   IF "PLC_Signals_DB".CH_NUMBER[0] THEN
       "PLC_Signals_DB".CH_NUMBER[1] := 0;
       "PLC_Signals_DB".CH_NUMBER[2] := 0;
       "PLC_Signals_DB".CH_NUMBER[3] := 0;
       "PLC_Signals_DB".CH_NUMBER[4] := 0;
       "PLC_Signals_DB".CH_NUMBER[5] := 0;
       "PLC_Signals_DB".CH_NUMBER[6] := 0;
       "PLC_Signals_DB".CH_NUMBER[7] := 0;
       "PLC_Signals_DB".CH_NUMBER[8] := 0;
       "PLC_Signals_DB".CH_NUMBER[9] := 0;
       "PLC_Signals_DB".CH_NUMBER[10] := 0;
       "PLC_Signals_DB".CH_NUMBER[11] := 0;
       "PLC_Signals_DB".CH_NUMBER[12] := 0;
       "PLC_Signals_DB".CH_NUMBER[13] := 0;
       "PLC_Signals_DB".CH_NUMBER[14] := 0;
       "PLC_Signals_DB".CH_NUMBER[15] := 0;
       "PLC_Signals_DB".CH_NUMBER[16] := 0;
       "PLC_Signals_DB".CH_NUMBER[17] := 0;
       "PLC_Signals_DB".CH_NUMBER[18] := 0;
       "PLC_Signals_DB".CH_NUMBER[19] := 0;
       "PLC_Signals_DB".CH_NUMBER[20] := 0;

       "DB_TST".CH_NUMBER := 0;
       "DB_TST".CH_NUMBER_OLD := "DB_TST".CH_NUMBER;
       "PLC_Signals_DB".CH_NUMBER[0] := 0;
   END_IF;

   CASE "DB_TST".CH_NUMBER OF
       1:
           IF "DB_TST".CH_NUMBER <> "DB_TST".CH_NUMBER_OLD THEN
               #Config_AI := #AI_2_0;
               "DB_TST".CH_NUMBER_OLD := "DB_TST".CH_NUMBER;
               ;
           END_IF;
           #Config_AI.ING_Value := #AI_2_0.ING_Value;
           #Config_AI.SCALED := #AI_2_0.SCALED;
           #Config_AI.State := #AI_2_0.State;
           #AI_2_0 := #Config_AI;
           ;
       2:
           IF "DB_TST".CH_NUMBER <> "DB_TST".CH_NUMBER_OLD THEN
               #Config_AI := #AI_2_1;
               "DB_TST".CH_NUMBER_OLD := "DB_TST".CH_NUMBER;
               ;
           END_IF;
           #Config_AI.ING_Value := #AI_2_1.ING_Value;
           #Config_AI.SCALED := #AI_2_1.SCALED;
           #Config_AI.State := #AI_2_1.State;
           #AI_2_1 := #Config_AI;
           ;
       3:
          IF "DB_TST".CH_NUMBER <> "DB_TST".CH_NUMBER_OLD THEN
               #Config_AI := #AI_2_2;
               "DB_TST".CH_NUMBER_OLD := "DB_TST".CH_NUMBER;
               ;
           END_IF;
           #Config_AI.ING_Value := #AI_2_2.ING_Value;
           #Config_AI.SCALED := #AI_2_2.SCALED;
           #Config_AI.State := #AI_2_2.State;
           #AI_2_2 := #Config_AI;
           ;
       4:
           IF "DB_TST".CH_NUMBER <> "DB_TST".CH_NUMBER_OLD THEN
               #Config_AI := #AI_2_3;
               "DB_TST".CH_NUMBER_OLD := "DB_TST".CH_NUMBER;
               ;
           END_IF;
           #Config_AI.ING_Value := #AI_2_3.ING_Value;
           #Config_AI.SCALED := #AI_2_3.SCALED;
           #Config_AI.State := #AI_2_3.State;
           #AI_2_3 := #Config_AI;
           ;
       5:
            IF "DB_TST".CH_NUMBER <> "DB_TST".CH_NUMBER_OLD THEN
               #Config_AI := #AI_2_4;
               "DB_TST".CH_NUMBER_OLD := "DB_TST".CH_NUMBER;
               ;
           END_IF;
           #Config_AI.ING_Value := #AI_2_4.ING_Value;
           #Config_AI.SCALED := #AI_2_4.SCALED;
           #Config_AI.State := #AI_2_4.State;
           #AI_2_4 := #Config_AI;
           ;
       6:
          IF "DB_TST".CH_NUMBER <> "DB_TST".CH_NUMBER_OLD THEN
               #Config_AI := #AI_2_5;
               "DB_TST".CH_NUMBER_OLD := "DB_TST".CH_NUMBER;
               ;
           END_IF;
           #Config_AI.ING_Value := #AI_2_5.ING_Value;
           #Config_AI.SCALED := #AI_2_5.SCALED;
           #Config_AI.State := #AI_2_5.State;
           #AI_2_5 := #Config_AI;
           ;
       7:
           IF "DB_TST".CH_NUMBER <> "DB_TST".CH_NUMBER_OLD THEN
               #Config_AI := #AI_2_6;
               "DB_TST".CH_NUMBER_OLD := "DB_TST".CH_NUMBER;
               ;
           END_IF;
           #Config_AI.ING_Value := #AI_2_6.ING_Value;
           #Config_AI.SCALED := #AI_2_6.SCALED;
           #Config_AI.State := #AI_2_6.State;
           #AI_2_6 := #Config_AI;
           ;
       8:
            IF "DB_TST".CH_NUMBER <> "DB_TST".CH_NUMBER_OLD THEN
               #Config_AI := #AI_2_7;
               "DB_TST".CH_NUMBER_OLD := "DB_TST".CH_NUMBER;
               ;
           END_IF;
           #Config_AI.ING_Value := #AI_2_7.ING_Value;
           #Config_AI.SCALED := #AI_2_7.SCALED;
           #Config_AI.State := #AI_2_7.State;
           #AI_2_7 := #Config_AI;
           ;
       9:
           IF "DB_TST".CH_NUMBER <> "DB_TST".CH_NUMBER_OLD THEN
               #Config_AI := #AI_3_0;
               "DB_TST".CH_NUMBER_OLD := "DB_TST".CH_NUMBER;
               ;
           END_IF;
           #Config_AI.ING_Value := #AI_3_0.ING_Value;
           #Config_AI.SCALED := #AI_3_0.SCALED;
           #Config_AI.State := #AI_3_0.State;
           #AI_3_0 := #Config_AI;
           ;
       10:
           IF "DB_TST".CH_NUMBER <> "DB_TST".CH_NUMBER_OLD THEN
               #Config_AI := #AI_3_1;
               "DB_TST".CH_NUMBER_OLD := "DB_TST".CH_NUMBER;
               ;
           END_IF;
           #Config_AI.ING_Value := #AI_3_1.ING_Value;
           #Config_AI.SCALED := #AI_3_1.SCALED;
           #Config_AI.State := #AI_3_1.State;
           #AI_3_1 := #Config_AI;
           ;
       11:
           IF "DB_TST".CH_NUMBER <> "DB_TST".CH_NUMBER_OLD THEN
               #Config_AI := #AI_3_2;
               "DB_TST".CH_NUMBER_OLD := "DB_TST".CH_NUMBER;
               ;
           END_IF;
           #Config_AI.ING_Value := #AI_3_2.ING_Value;
           #Config_AI.SCALED := #AI_3_2.SCALED;
           #Config_AI.State := #AI_3_2.State;
           #AI_3_2 := #Config_AI;
           ;
       12:
           IF "DB_TST".CH_NUMBER <> "DB_TST".CH_NUMBER_OLD THEN
               #Config_AI := #AI_3_3;
               "DB_TST".CH_NUMBER_OLD := "DB_TST".CH_NUMBER;
               ;
           END_IF;
           #Config_AI.ING_Value := #AI_3_3.ING_Value;
           #Config_AI.SCALED := #AI_3_3.SCALED;
           #Config_AI.State := #AI_3_3.State;
           #AI_3_3 := #Config_AI;
           ;
       13:
           IF "DB_TST".CH_NUMBER <> "DB_TST".CH_NUMBER_OLD THEN
               #Config_AI := #AI_3_4;
               "DB_TST".CH_NUMBER_OLD := "DB_TST".CH_NUMBER;
               ;
           END_IF;
           #Config_AI.ING_Value := #AI_3_4.ING_Value;
           #Config_AI.SCALED := #AI_3_4.SCALED;
           #Config_AI.State := #AI_3_4.State;
           #AI_3_4 := #Config_AI;
           ;
       14:
           IF "DB_TST".CH_NUMBER <> "DB_TST".CH_NUMBER_OLD THEN
               #Config_AI := #AI_3_5;
               "DB_TST".CH_NUMBER_OLD := "DB_TST".CH_NUMBER;
               ;
           END_IF;
           #Config_AI.ING_Value := #AI_3_5.ING_Value;
           #Config_AI.SCALED := #AI_3_5.SCALED;
           #Config_AI.State := #AI_3_5.State;
           #AI_3_5 := #Config_AI;
           ;
       15:
           IF "DB_TST".CH_NUMBER <> "DB_TST".CH_NUMBER_OLD THEN
               #Config_AI := #AI_3_6;
               "DB_TST".CH_NUMBER_OLD := "DB_TST".CH_NUMBER;
               ;
           END_IF;
           #Config_AI.ING_Value := #AI_3_6.ING_Value;
           #Config_AI.SCALED := #AI_3_6.SCALED;
           #Config_AI.State := #AI_3_6.State;
           #AI_3_6 := #Config_AI;
           ;
       16:
           IF "DB_TST".CH_NUMBER <> "DB_TST".CH_NUMBER_OLD THEN
               #Config_AI := #AI_3_7;
               "DB_TST".CH_NUMBER_OLD := "DB_TST".CH_NUMBER;
               ;
           END_IF;
           #Config_AI.ING_Value := #AI_3_7.ING_Value;
           #Config_AI.SCALED := #AI_3_7.SCALED;
           #Config_AI.State := #AI_3_7.State;
           #AI_3_7 := #Config_AI;
           ;
       ELSE  // Statement section ELSE
           ;
   END_CASE;
END_FUNCTION

FUNCTION "AI" : Void   // FC24, LAD
{ S7_Optimized_Access := 'TRUE' }
VERSION : 0.1
   VAR_IN_OUT
      AI : Struct   // ????????? ? AI
         Hihi_Value : Real;   // True
         High_Value : Real;   // True
         Low_Value : Real;   // True
         Lolo_Value : Real;   // True
         MIN_Current : Real;   // True
         MAX_Current : Real;   // True
         MAX_Value : Real;   // True
         MIN_Value : Real;   // True
         Underflow_RAW : Real;   // True
         Overflow_RAW : Real;   // True
         SCALED : Real;   // True
         ING_Value : Real;   // True
         Manual_Value : Real;   // True
         Alarm_Delay : Int;   // True
         Warning_Delay : Int;   // True
         AVG_Delay : Real;   // True
         Underflow_Delay : Int;   // True
         Overflow_Delay : Int;   // True
         StateHMI : Int;
         State : Word;   // True
         Modeee : Word;   // True
         bools : Word;   // True
         AI_RAW_MIN : Int;   // True
         AI_RAW_MAX : Int;   // True
         Hihi_EN : Bool;   // True
         High_EN : Bool;   // True
         Low_En : Bool;   // True
         Lolo_EN : Bool;   // True
      END_STRUCT;
      AI_RAW : Int;   // ???????? ??? ?? ?????
      Hihi_TImer : IEC_TIMER;
      High_Timer : IEC_TIMER;
      Low_Timer : IEC_TIMER;
      Lolo_Timer : IEC_TIMER;
      WB_Timer : IEC_TIMER;
      OVerflow_Timer : IEC_TIMER;
   END_VAR
   VAR_TEMP
      Hihi_Int : Bool;   // ????????????? ???????????? ??????? Hihi ??? ?????????? ???????? ?????????
      High_Int : Bool;   // ????????????? ???????????? ??????? High ??? ?????????? ???????? ?????????
      Low_Int : Bool;   // ????????????? ???????????? ??????? Low ??? ?????????? ???????? ?????????
      Lolo_Int : Bool;   // ????????????? ???????????? ??????? Lolo ??? ?????????? ???????? ?????????
      Scaled_4_20mA : Real;   // ???????? ???? ?? ?????, ???????????????? ? 4-20??
      WB_Int : Bool;   // ????????????? ????????????? ?????? ???????
      Last_value : Real;   // ???????? ??? FailSafe_Mode
      count : Int;   // ?????????? ???????? ??? ??????????
      time_int : Int;   // ????? ? INT
      current_count : Int;   // ??????? ?????????? ???????? ??? ??????????
      summ_AVG_Value : Real;   // ????? ???????? ??? ??????????
      tmp_scaled : Real;   // ???????????????? ???????? ??? ??????????
      Overflow_int : Bool;   // ??????????????? ???????????? ????????????? ??????? <
      Underflow_int : Bool;   // ??????????????? ???????????? ????????????? ??????? >
      AVG_Delay_real : Real;
      Alarm_Delay_int : Time;
      Warning_Delay_int : Time;
      Underflow_Delay_int : Time;
      Overflow_Delay_int : Time;
      TMP_ING_Value : Real;
      et1 : Time;
      et2 : Time;
      et3 : Time;
      et4 : Time;
      et5 : Time;
      et6 : Time;
      ust_avg_up : Real;
      ust_avg_down : Real;
   END_VAR
   VAR CONSTANT
      AI_Time : Int := 250;   // ????? ?????? AI (??)
   END_VAR
   VAR_TEMP   // added for the SCL form of the ladder/FBD networks
      _w1 : Bool;
      _w2 : Bool;
      _w3 : Bool;
      _w4 : Bool;
      _w5 : Bool;
      _w6 : Bool;
      _w7 : Bool;
      _w8 : Bool;
      _w9 : Bool;
      _w10 : Bool;
      _w11 : Bool;
      _w12 : Bool;
      _w13 : Bool;
      _w14 : Bool;
      _w15 : Bool;
   END_VAR
BEGIN

REGION Network 1: Пересчет времени
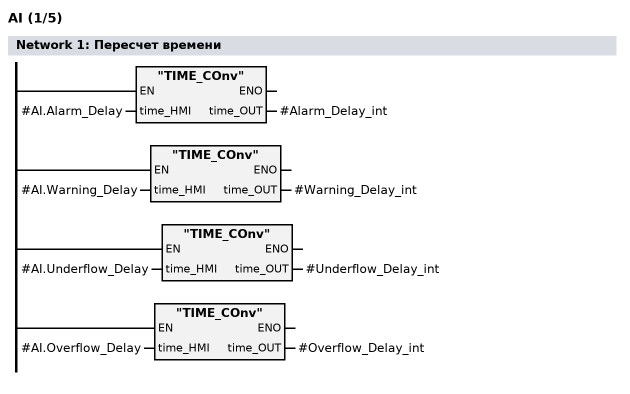
   RUNG wire#powerrail
      "TIME_COnv"(time_HMI := #AI.Alarm_Delay, time_OUT => #Alarm_Delay_int)
   END_RUNG
   RUNG wire#powerrail
      "TIME_COnv"(time_HMI := #AI.Warning_Delay, time_OUT => #Warning_Delay_int)
   END_RUNG
   RUNG wire#powerrail
      "TIME_COnv"(time_HMI := #AI.Underflow_Delay, time_OUT => #Underflow_Delay_int)
   END_RUNG
   RUNG wire#powerrail
      "TIME_COnv"(time_HMI := #AI.Overflow_Delay, time_OUT => #Overflow_Delay_int)
   END_RUNG
   // the same network as SCL:
   "TIME_COnv"(time_HMI := #AI.Alarm_Delay, time_OUT => #Alarm_Delay_int);
   "TIME_COnv"(time_HMI := #AI.Warning_Delay, time_OUT => #Warning_Delay_int);
   "TIME_COnv"(time_HMI := #AI.Underflow_Delay, time_OUT => #Underflow_Delay_int);
   "TIME_COnv"(time_HMI := #AI.Overflow_Delay, time_OUT => #Overflow_Delay_int);
END_REGION

REGION Network 2: авто конвертация в инж. и физ. значение
   // Автоматическая обработка сигналов
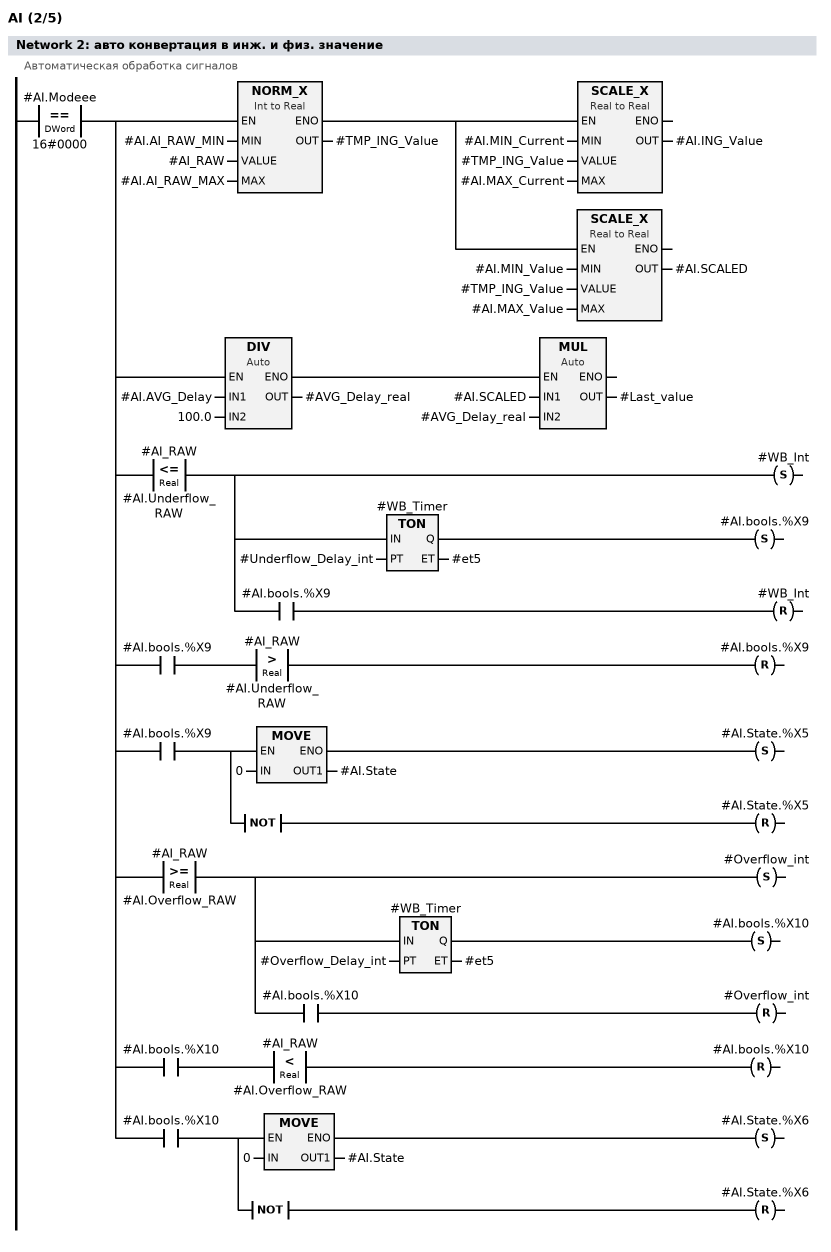
   // ENO of a box is taken as its EN; it also drops when the box reports an error
   #_w1 := #AI.Modeee = 16#0000;
   IF #_w1 THEN
       #TMP_ING_Value := NORM_X(MIN := #AI.AI_RAW_MIN, VALUE := #AI_RAW, MAX := #AI.AI_RAW_MAX);
       #AI.ING_Value := SCALE_X(MIN := #AI.MIN_Current, VALUE := #TMP_ING_Value, MAX := #AI.MAX_Current);
       #AI.SCALED := SCALE_X(MIN := #AI.MIN_Value, VALUE := #TMP_ING_Value, MAX := #AI.MAX_Value);
       #AVG_Delay_real := #AI.AVG_Delay / 100.0;
       #Last_value := #AI.SCALED * #AVG_Delay_real;
   END_IF;
   #_w2 := #_w1 AND (#AI_RAW <= #AI.Underflow_RAW);
   IF #_w2 THEN #WB_Int := TRUE; END_IF;
   #WB_Timer.TON(IN := #_w2, PT := #Underflow_Delay_int, ET => #et5);
   IF #WB_Timer.Q THEN #AI.bools.%X9 := TRUE; END_IF;
   IF #_w2 AND #AI.bools.%X9 THEN #WB_Int := FALSE; END_IF;
   IF #_w1 AND #AI.bools.%X9 AND (#AI_RAW > #AI.Underflow_RAW) THEN #AI.bools.%X9 := FALSE; END_IF;
   #_w3 := #_w1 AND #AI.bools.%X9;
   IF #_w3 THEN
       #AI.State := 0;
       #AI.State.%X5 := TRUE;
   END_IF;
   IF NOT #_w3 THEN #AI.State.%X5 := FALSE; END_IF;
   #_w4 := #_w1 AND (#AI_RAW >= #AI.Overflow_RAW);
   IF #_w4 THEN #Overflow_int := TRUE; END_IF;
   #WB_Timer.TON(IN := #_w4, PT := #Overflow_Delay_int, ET => #et5);
   IF #WB_Timer.Q THEN #AI.bools.%X10 := TRUE; END_IF;
   IF #_w4 AND #AI.bools.%X10 THEN #Overflow_int := FALSE; END_IF;
   IF #_w1 AND #AI.bools.%X10 AND (#AI_RAW < #AI.Overflow_RAW) THEN #AI.bools.%X10 := FALSE; END_IF;
   #_w5 := #_w1 AND #AI.bools.%X10;
   IF #_w5 THEN
       #AI.State := 0;
       #AI.State.%X6 := TRUE;
   END_IF;
   IF NOT #_w5 THEN #AI.State.%X6 := FALSE; END_IF;
END_REGION

REGION Network 3: ручной ввод и ремонт, при это ток вседа равен 4мА, чтобы обрыв не вылетал
   // ремонт или ручной ввод
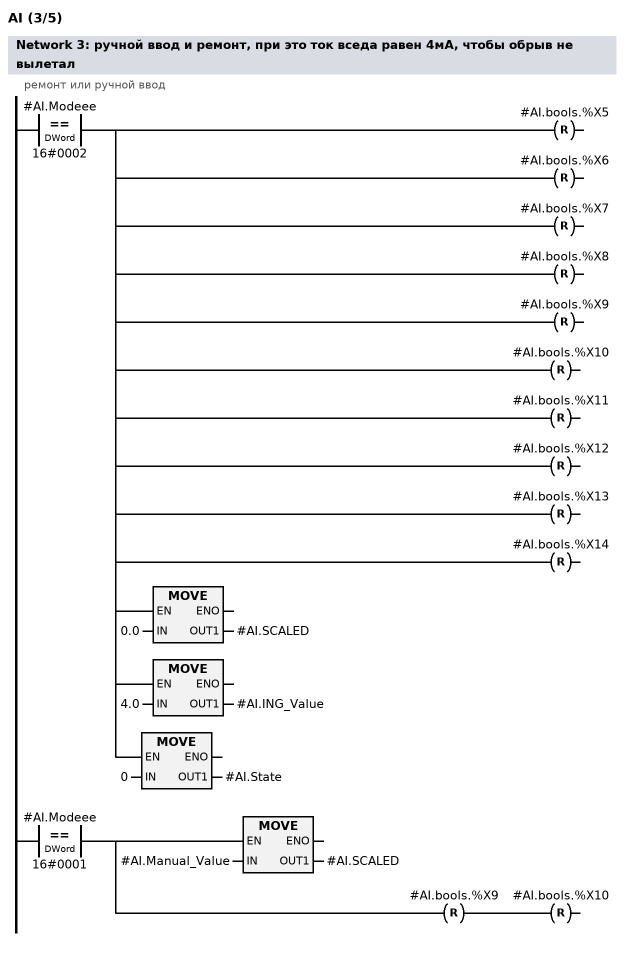
   RUNG wire#powerrail
      { S7_Templates := "SrcType := DWord" } EQ_Contact(in1 := #AI.Modeee, in2 := 16#0002)
      wire#w1
      R_Coil( #AI.bools.%X5 )
   END_RUNG
   RUNG wire#w1
      R_Coil( #AI.bools.%X6 )
   END_RUNG
   RUNG wire#w1
      R_Coil( #AI.bools.%X7 )
   END_RUNG
   RUNG wire#w1
      R_Coil( #AI.bools.%X8 )
   END_RUNG
   RUNG wire#w1
      R_Coil( #AI.bools.%X9 )
   END_RUNG
   RUNG wire#w1
      R_Coil( #AI.bools.%X10 )
   END_RUNG
   RUNG wire#w1
      R_Coil( #AI.bools.%X11 )
   END_RUNG
   RUNG wire#w1
      R_Coil( #AI.bools.%X12 )
   END_RUNG
   RUNG wire#w1
      R_Coil( #AI.bools.%X13 )
   END_RUNG
   RUNG wire#w1
      R_Coil( #AI.bools.%X14 )
   END_RUNG
   RUNG wire#w1
      { S7_GenerateENO := "TRUE" } Move(in := 0.0, out1 => #AI.SCALED)
   END_RUNG
   RUNG wire#w1
      { S7_GenerateENO := "TRUE" } Move(in := 4.0, out1 => #AI.ING_Value)
   END_RUNG
   RUNG wire#w1
      { S7_GenerateENO := "TRUE" } Move(in := 0, out1 => #AI.State)
   END_RUNG
   RUNG wire#powerrail
      { S7_Templates := "SrcType := DWord" } EQ_Contact(in1 := #AI.Modeee, in2 := 16#0001)
      wire#w2
      { S7_GenerateENO := "TRUE" } Move(in := #AI.Manual_Value, out1 => #AI.SCALED)
   END_RUNG
   RUNG wire#w2
      R_Coil( #AI.bools.%X9 )
      R_Coil( #AI.bools.%X10 )
   END_RUNG
   // the same network as SCL:
   IF #AI.Modeee = 16#0002 THEN
       #AI.bools.%X5 := FALSE;
       #AI.bools.%X6 := FALSE;
       #AI.bools.%X7 := FALSE;
       #AI.bools.%X8 := FALSE;
       #AI.bools.%X9 := FALSE;
       #AI.bools.%X10 := FALSE;
       #AI.bools.%X11 := FALSE;
       #AI.bools.%X12 := FALSE;
       #AI.bools.%X13 := FALSE;
       #AI.bools.%X14 := FALSE;
       #AI.SCALED := 0.0;
       #AI.ING_Value := 4.0;
       #AI.State := 0;
   END_IF;
   IF #AI.Modeee = 16#0001 THEN
       #AI.SCALED := #AI.Manual_Value;
       #AI.bools.%X9 := FALSE;
       #AI.bools.%X10 := FALSE;
   END_IF;
END_REGION

REGION Network 4: уставки
   // Автоматическая обработка сигналов
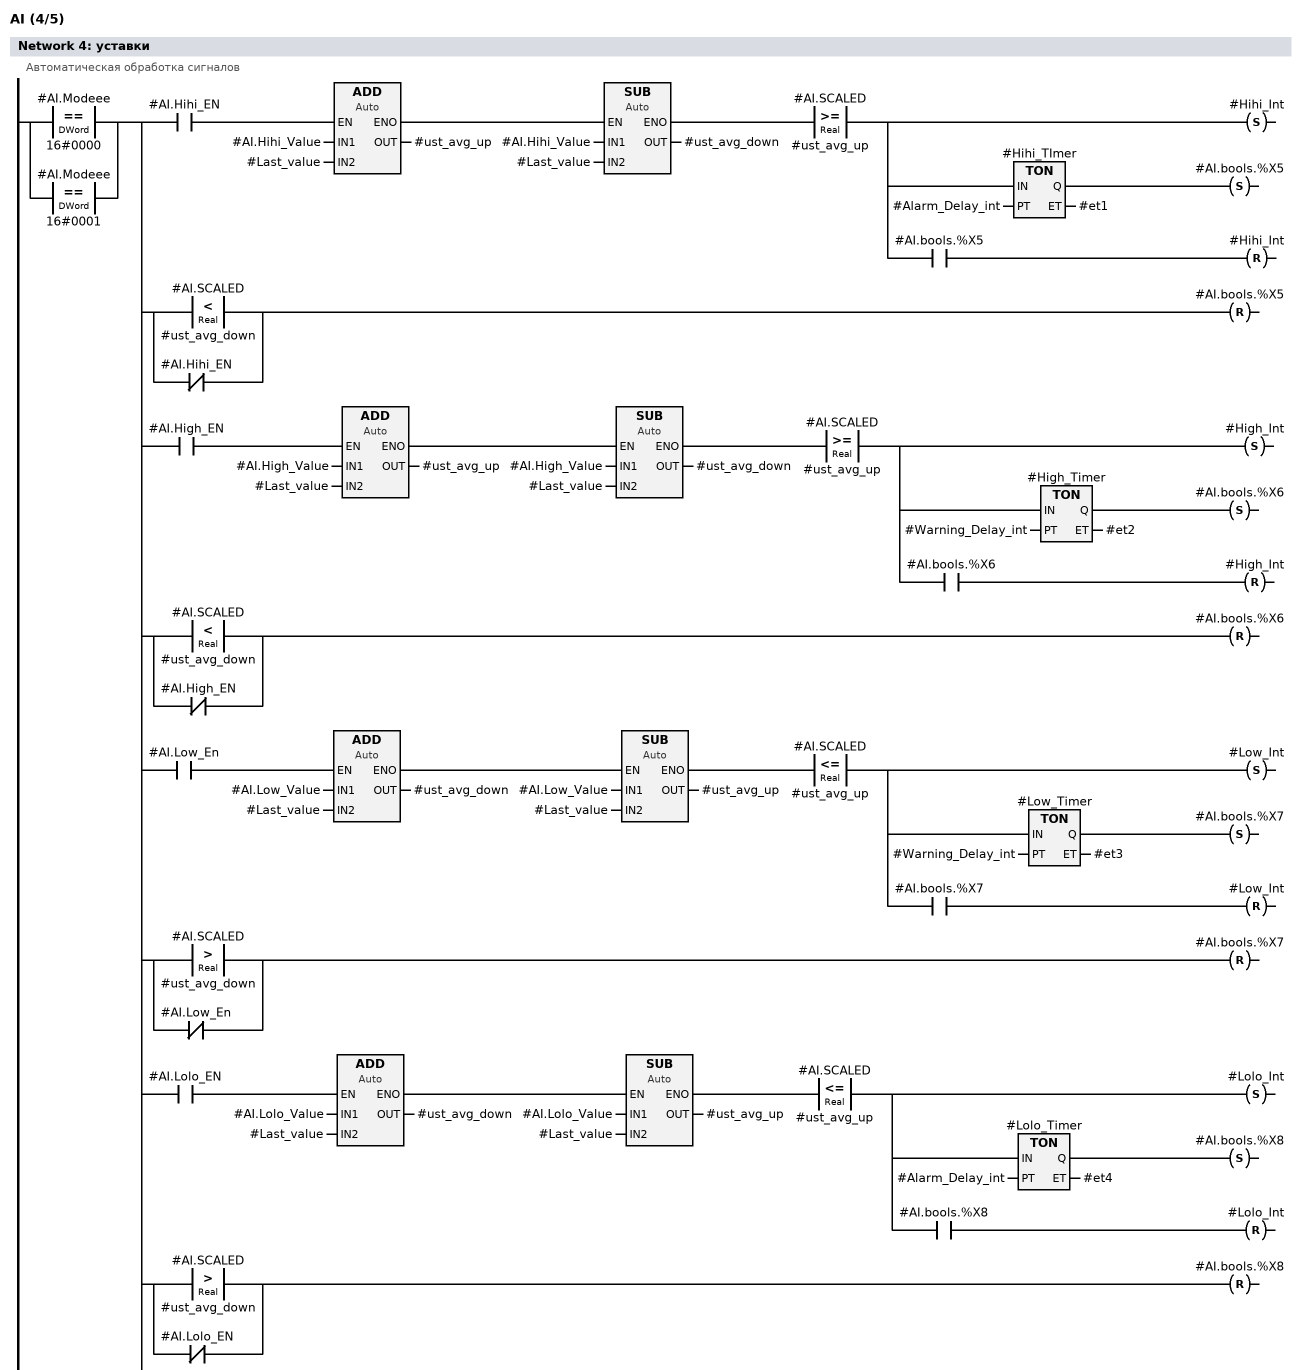
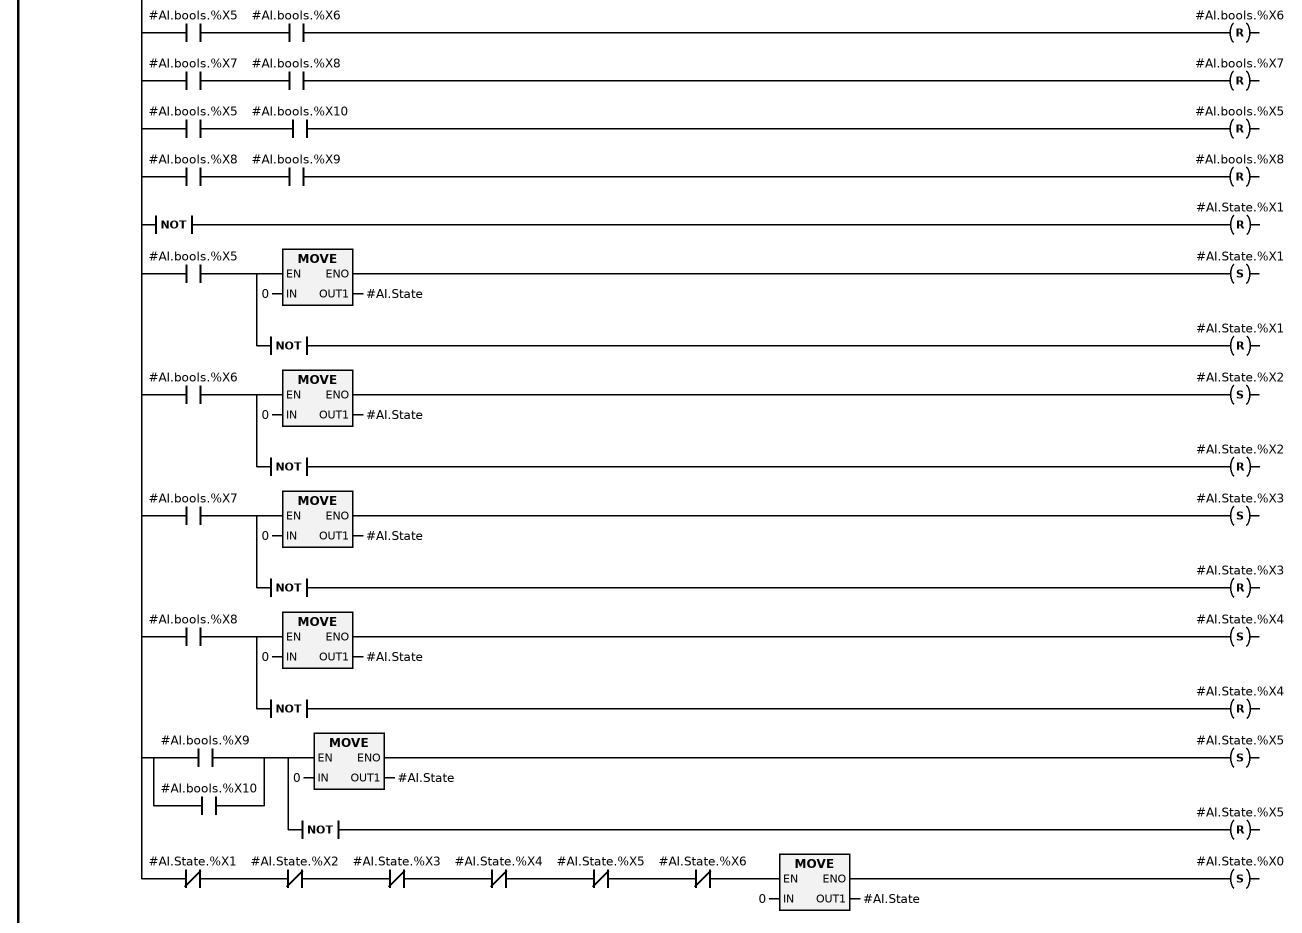
   // ENO of a box is taken as its EN; it also drops when the box reports an error
   #_w1 := (#AI.Modeee = 16#0000) OR (#AI.Modeee = 16#0001);
   #_w2 := #_w1 AND #AI.Hihi_EN;
   IF #_w2 THEN
       #ust_avg_up := #AI.Hihi_Value + #Last_value;
       #ust_avg_down := #AI.Hihi_Value - #Last_value;
   END_IF;
   #_w3 := #_w2 AND (#AI.SCALED >= #ust_avg_up);
   IF #_w3 THEN #Hihi_Int := TRUE; END_IF;
   #Hihi_TImer.TON(IN := #_w3, PT := #Alarm_Delay_int, ET => #et1);
   IF #Hihi_TImer.Q THEN #AI.bools.%X5 := TRUE; END_IF;
   IF #_w3 AND #AI.bools.%X5 THEN #Hihi_Int := FALSE; END_IF;
   IF #_w1 AND ((#AI.SCALED < #ust_avg_down) OR NOT #AI.Hihi_EN) THEN #AI.bools.%X5 := FALSE; END_IF;
   #_w4 := #_w1 AND #AI.High_EN;
   IF #_w4 THEN
       #ust_avg_up := #AI.High_Value + #Last_value;
       #ust_avg_down := #AI.High_Value - #Last_value;
   END_IF;
   #_w5 := #_w4 AND (#AI.SCALED >= #ust_avg_up);
   IF #_w5 THEN #High_Int := TRUE; END_IF;
   #High_Timer.TON(IN := #_w5, PT := #Warning_Delay_int, ET => #et2);
   IF #High_Timer.Q THEN #AI.bools.%X6 := TRUE; END_IF;
   IF #_w5 AND #AI.bools.%X6 THEN #High_Int := FALSE; END_IF;
   IF #_w1 AND ((#AI.SCALED < #ust_avg_down) OR NOT #AI.High_EN) THEN #AI.bools.%X6 := FALSE; END_IF;
   #_w6 := #_w1 AND #AI.Low_En;
   IF #_w6 THEN
       #ust_avg_down := #AI.Low_Value + #Last_value;
       #ust_avg_up := #AI.Low_Value - #Last_value;
   END_IF;
   #_w7 := #_w6 AND (#AI.SCALED <= #ust_avg_up);
   IF #_w7 THEN #Low_Int := TRUE; END_IF;
   #Low_Timer.TON(IN := #_w7, PT := #Warning_Delay_int, ET => #et3);
   IF #Low_Timer.Q THEN #AI.bools.%X7 := TRUE; END_IF;
   IF #_w7 AND #AI.bools.%X7 THEN #Low_Int := FALSE; END_IF;
   IF #_w1 AND ((#AI.SCALED > #ust_avg_down) OR NOT #AI.Low_En) THEN #AI.bools.%X7 := FALSE; END_IF;
   #_w8 := #_w1 AND #AI.Lolo_EN;
   IF #_w8 THEN
       #ust_avg_down := #AI.Lolo_Value + #Last_value;
       #ust_avg_up := #AI.Lolo_Value - #Last_value;
   END_IF;
   #_w9 := #_w8 AND (#AI.SCALED <= #ust_avg_up);
   IF #_w9 THEN #Lolo_Int := TRUE; END_IF;
   #Lolo_Timer.TON(IN := #_w9, PT := #Alarm_Delay_int, ET => #et4);
   IF #Lolo_Timer.Q THEN #AI.bools.%X8 := TRUE; END_IF;
   IF #_w9 AND #AI.bools.%X8 THEN #Lolo_Int := FALSE; END_IF;
   IF #_w1 AND ((#AI.SCALED > #ust_avg_down) OR NOT #AI.Lolo_EN) THEN #AI.bools.%X8 := FALSE; END_IF;
   IF #_w1 AND #AI.bools.%X5 AND #AI.bools.%X6 THEN #AI.bools.%X6 := FALSE; END_IF;
   IF #_w1 AND #AI.bools.%X7 AND #AI.bools.%X8 THEN #AI.bools.%X7 := FALSE; END_IF;
   IF #_w1 AND #AI.bools.%X5 AND #AI.bools.%X10 THEN #AI.bools.%X5 := FALSE; END_IF;
   IF #_w1 AND #AI.bools.%X8 AND #AI.bools.%X9 THEN #AI.bools.%X8 := FALSE; END_IF;
   IF NOT #_w1 THEN #AI.State.%X1 := FALSE; END_IF;
   #_w10 := #_w1 AND #AI.bools.%X5;
   IF #_w10 THEN
       #AI.State := 0;
       #AI.State.%X1 := TRUE;
   END_IF;
   IF NOT #_w10 THEN #AI.State.%X1 := FALSE; END_IF;
   #_w11 := #_w1 AND #AI.bools.%X6;
   IF #_w11 THEN
       #AI.State := 0;
       #AI.State.%X2 := TRUE;
   END_IF;
   IF NOT #_w11 THEN #AI.State.%X2 := FALSE; END_IF;
   #_w12 := #_w1 AND #AI.bools.%X7;
   IF #_w12 THEN
       #AI.State := 0;
       #AI.State.%X3 := TRUE;
   END_IF;
   IF NOT #_w12 THEN #AI.State.%X3 := FALSE; END_IF;
   #_w13 := #_w1 AND #AI.bools.%X8;
   IF #_w13 THEN
       #AI.State := 0;
       #AI.State.%X4 := TRUE;
   END_IF;
   IF NOT #_w13 THEN #AI.State.%X4 := FALSE; END_IF;
   #_w14 := #_w1 AND (#AI.bools.%X9 OR #AI.bools.%X10);
   IF #_w14 THEN
       #AI.State := 0;
       #AI.State.%X5 := TRUE;
   END_IF;
   IF NOT #_w14 THEN #AI.State.%X5 := FALSE; END_IF;
   #_w15 := #_w1 AND NOT #AI.State.%X1 AND NOT #AI.State.%X2 AND NOT #AI.State.%X3 AND NOT #AI.State.%X4 AND NOT #AI.State.%X5 AND NOT #AI.State.%X6;
   IF #_w15 THEN
       #AI.State := 0;
       #AI.State.%X0 := TRUE;
   END_IF;
END_REGION

REGION Network 5
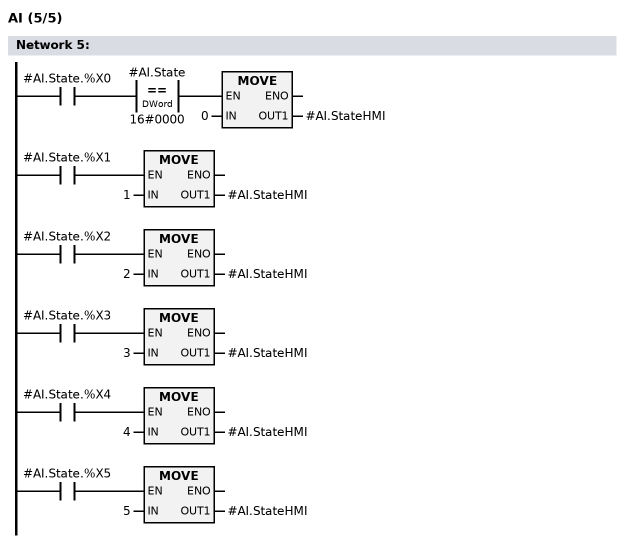
   RUNG wire#powerrail
      Contact( #AI.State.%X0 )
      { S7_Templates := "SrcType := DWord" } EQ_Contact(in1 := #AI.State, in2 := 16#0000)
      Move(in := 0, out1 => #AI.StateHMI)
   END_RUNG
   RUNG wire#powerrail
      Contact( #AI.State.%X1 )
      Move(in := 1, out1 => #AI.StateHMI)
   END_RUNG
   RUNG wire#powerrail
      Contact( #AI.State.%X2 )
      Move(in := 2, out1 => #AI.StateHMI)
   END_RUNG
   RUNG wire#powerrail
      Contact( #AI.State.%X3 )
      Move(in := 3, out1 => #AI.StateHMI)
   END_RUNG
   RUNG wire#powerrail
      Contact( #AI.State.%X4 )
      Move(in := 4, out1 => #AI.StateHMI)
   END_RUNG
   RUNG wire#powerrail
      Contact( #AI.State.%X5 )
      Move(in := 5, out1 => #AI.StateHMI)
   END_RUNG
   // the same network as SCL:
   IF #AI.State.%X0 AND (#AI.State = 16#0000) THEN #AI.StateHMI := 0; END_IF;
   IF #AI.State.%X1 THEN #AI.StateHMI := 1; END_IF;
   IF #AI.State.%X2 THEN #AI.StateHMI := 2; END_IF;
   IF #AI.State.%X3 THEN #AI.StateHMI := 3; END_IF;
   IF #AI.State.%X4 THEN #AI.StateHMI := 4; END_IF;
   IF #AI.State.%X5 THEN #AI.StateHMI := 5; END_IF;
END_REGION
END_FUNCTION

FUNCTION "TIME_COnv" : Void   // FC26, SCL
{ S7_Optimized_Access := 'TRUE' }
VERSION : 0.1
   VAR_INPUT
      time_HMI : Int;
   END_VAR
   VAR_OUTPUT
      time_OUT : Time;
   END_VAR
   VAR_TEMP
      "DINT" : DInt;
      t_DINT : DInt;
   END_VAR
BEGIN
   #t_DINT := INT_TO_DINT(#time_HMI);
   #"DINT" := #t_DINT * 1000;

   #time_OUT := T_CONV(#"DINT");
END_FUNCTION

ORGANIZATION_BLOCK "Main"   // OB1, LAD, ProgramCycle
TITLE = "Main Program Sweep (Cycle)"
{ S7_Optimized_Access := 'TRUE' }
VERSION : 0.1
   VAR_INPUT
      Initial_Call : Bool;   // Initial call of this OB
      Remanence : Bool;   // =True, if remanent data are available
   END_VAR
   VAR_TEMP
      alarm_nmsh : Bool;
      zp_nmsh : Bool;
      alarm_nd_1 : Bool;
      zp_nd_1 : Bool;
      alarm_nd_2 : Bool;
      zp_nd_2 : Bool;
   END_VAR
   VAR_TEMP   // added for the SCL form of the ladder/FBD networks
      _w1 : Bool;
   END_VAR
BEGIN

REGION Network 1: Настройка аналогов с панели
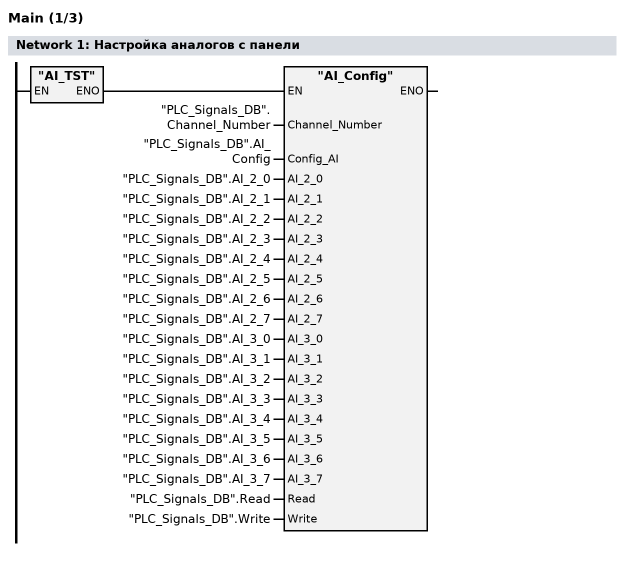
   RUNG wire#powerrail
      "AI_TST"()
      "AI_Config"(Channel_Number := "PLC_Signals_DB".Channel_Number, Config_AI := "PLC_Signals_DB".AI_Config, AI_2_0 := "PLC_Signals_DB".AI_2_0, AI_2_1 := "PLC_Signals_DB".AI_2_1, AI_2_2 := "PLC_Signals_DB".AI_2_2, AI_2_3 := "PLC_Signals_DB".AI_2_3, AI_2_4 := "PLC_Signals_DB".AI_2_4, AI_2_5 := "PLC_Signals_DB".AI_2_5, AI_2_6 := "PLC_Signals_DB".AI_2_6, AI_2_7 := "PLC_Signals_DB".AI_2_7, AI_3_0 := "PLC_Signals_DB".AI_3_0, AI_3_1 := "PLC_Signals_DB".AI_3_1, AI_3_2 := "PLC_Signals_DB".AI_3_2, AI_3_3 := "PLC_Signals_DB".AI_3_3, AI_3_4 := "PLC_Signals_DB".AI_3_4, AI_3_5 := "PLC_Signals_DB".AI_3_5, AI_3_6 := "PLC_Signals_DB".AI_3_6, AI_3_7 := "PLC_Signals_DB".AI_3_7, Read := "PLC_Signals_DB".Read, Write := "PLC_Signals_DB".Write)
   END_RUNG
   // the same network as SCL:
   "AI_TST"(ENO => #_w1);
   IF #_w1 THEN
       "AI_Config"(Channel_Number := "PLC_Signals_DB".Channel_Number,
                   Config_AI := "PLC_Signals_DB".AI_Config,
                   AI_2_0 := "PLC_Signals_DB".AI_2_0,
                   AI_2_1 := "PLC_Signals_DB".AI_2_1,
                   AI_2_2 := "PLC_Signals_DB".AI_2_2,
                   AI_2_3 := "PLC_Signals_DB".AI_2_3,
                   AI_2_4 := "PLC_Signals_DB".AI_2_4,
                   AI_2_5 := "PLC_Signals_DB".AI_2_5,
                   AI_2_6 := "PLC_Signals_DB".AI_2_6,
                   AI_2_7 := "PLC_Signals_DB".AI_2_7,
                   AI_3_0 := "PLC_Signals_DB".AI_3_0,
                   AI_3_1 := "PLC_Signals_DB".AI_3_1,
                   AI_3_2 := "PLC_Signals_DB".AI_3_2,
                   AI_3_3 := "PLC_Signals_DB".AI_3_3,
                   AI_3_4 := "PLC_Signals_DB".AI_3_4,
                   AI_3_5 := "PLC_Signals_DB".AI_3_5,
                   AI_3_6 := "PLC_Signals_DB".AI_3_6,
                   AI_3_7 := "PLC_Signals_DB".AI_3_7,
                   Read := "PLC_Signals_DB".Read,
                   Write := "PLC_Signals_DB".Write);
   END_IF;
END_REGION

REGION Network 2: Горелка
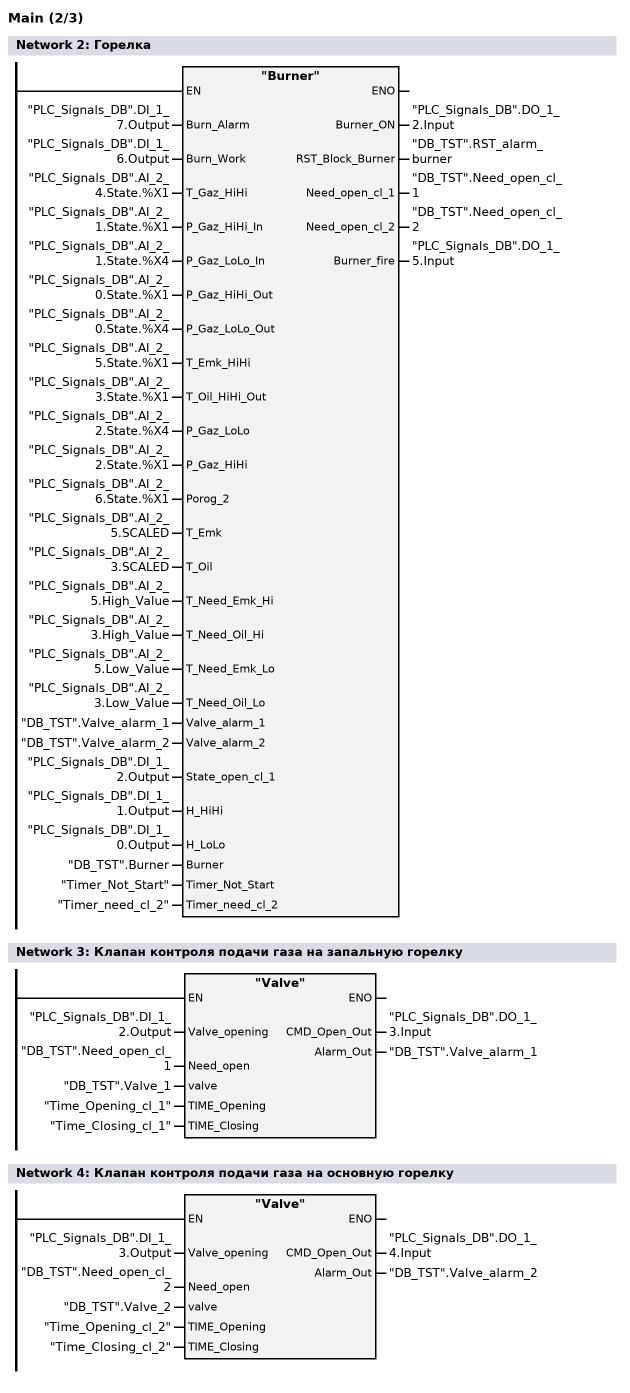
   RUNG wire#powerrail
      "Burner"(Burn_Alarm := "PLC_Signals_DB".DI_1_7.Output, Burn_Work := "PLC_Signals_DB".DI_1_6.Output, T_Gaz_HiHi := "PLC_Signals_DB".AI_2_4.State.%X1, P_Gaz_HiHi_In := "PLC_Signals_DB".AI_2_1.State.%X1, P_Gaz_LoLo_In := "PLC_Signals_DB".AI_2_1.State.%X4, P_Gaz_HiHi_Out := "PLC_Signals_DB".AI_2_0.State.%X1, P_Gaz_LoLo_Out := "PLC_Signals_DB".AI_2_0.State.%X4, T_Emk_HiHi := "PLC_Signals_DB".AI_2_5.State.%X1, T_Oil_HiHi_Out := "PLC_Signals_DB".AI_2_3.State.%X1, P_Gaz_LoLo := "PLC_Signals_DB".AI_2_2.State.%X4, P_Gaz_HiHi := "PLC_Signals_DB".AI_2_2.State.%X1, Porog_2 := "PLC_Signals_DB".AI_2_6.State.%X1, T_Emk := "PLC_Signals_DB".AI_2_5.SCALED, T_Oil := "PLC_Signals_DB".AI_2_3.SCALED, T_Need_Emk_Hi := "PLC_Signals_DB".AI_2_5.High_Value, T_Need_Oil_Hi := "PLC_Signals_DB".AI_2_3.High_Value, T_Need_Emk_Lo := "PLC_Signals_DB".AI_2_5.Low_Value, T_Need_Oil_Lo := "PLC_Signals_DB".AI_2_3.Low_Value, Valve_alarm_1 := "DB_TST".Valve_alarm_1, Valve_alarm_2 := "DB_TST".Valve_alarm_2, State_open_cl_1 := "PLC_Signals_DB".DI_1_2.Output, H_HiHi := "PLC_Signals_DB".DI_1_1.Output, H_LoLo := "PLC_Signals_DB".DI_1_0.Output, Burner := "DB_TST".Burner, Timer_Not_Start := "Timer_Not_Start", Timer_need_cl_2 := "Timer_need_cl_2", Burner_ON => "PLC_Signals_DB".DO_1_2.Input, RST_Block_Burner => "DB_TST".RST_alarm_burner, Need_open_cl_1 => "DB_TST".Need_open_cl_1, Need_open_cl_2 => "DB_TST".Need_open_cl_2, Burner_fire => "PLC_Signals_DB".DO_1_5.Input)
   END_RUNG
   // the same network as SCL:
   "Burner"(Burn_Alarm := "PLC_Signals_DB".DI_1_7.Output,
            Burn_Work := "PLC_Signals_DB".DI_1_6.Output,
            T_Gaz_HiHi := "PLC_Signals_DB".AI_2_4.State.%X1,
            P_Gaz_HiHi_In := "PLC_Signals_DB".AI_2_1.State.%X1,
            P_Gaz_LoLo_In := "PLC_Signals_DB".AI_2_1.State.%X4,
            P_Gaz_HiHi_Out := "PLC_Signals_DB".AI_2_0.State.%X1,
            P_Gaz_LoLo_Out := "PLC_Signals_DB".AI_2_0.State.%X4,
            T_Emk_HiHi := "PLC_Signals_DB".AI_2_5.State.%X1,
            T_Oil_HiHi_Out := "PLC_Signals_DB".AI_2_3.State.%X1,
            P_Gaz_LoLo := "PLC_Signals_DB".AI_2_2.State.%X4,
            P_Gaz_HiHi := "PLC_Signals_DB".AI_2_2.State.%X1,
            Porog_2 := "PLC_Signals_DB".AI_2_6.State.%X1,
            T_Emk := "PLC_Signals_DB".AI_2_5.SCALED,
            T_Oil := "PLC_Signals_DB".AI_2_3.SCALED,
            T_Need_Emk_Hi := "PLC_Signals_DB".AI_2_5.High_Value,
            T_Need_Oil_Hi := "PLC_Signals_DB".AI_2_3.High_Value,
            T_Need_Emk_Lo := "PLC_Signals_DB".AI_2_5.Low_Value,
            T_Need_Oil_Lo := "PLC_Signals_DB".AI_2_3.Low_Value,
            Valve_alarm_1 := "DB_TST".Valve_alarm_1,
            Valve_alarm_2 := "DB_TST".Valve_alarm_2,
            State_open_cl_1 := "PLC_Signals_DB".DI_1_2.Output,
            H_HiHi := "PLC_Signals_DB".DI_1_1.Output,
            H_LoLo := "PLC_Signals_DB".DI_1_0.Output,
            Burner := "DB_TST".Burner,
            Timer_Not_Start := "Timer_Not_Start",
            Timer_need_cl_2 := "Timer_need_cl_2",
            Burner_ON => "PLC_Signals_DB".DO_1_2.Input,
            RST_Block_Burner => "DB_TST".RST_alarm_burner,
            Need_open_cl_1 => "DB_TST".Need_open_cl_1,
            Need_open_cl_2 => "DB_TST".Need_open_cl_2,
            Burner_fire => "PLC_Signals_DB".DO_1_5.Input);
END_REGION

REGION Network 3: Клапан контроля подачи газа на запальную горелку
   RUNG wire#powerrail
      "Valve"(Valve_opening := "PLC_Signals_DB".DI_1_2.Output, Need_open := "DB_TST".Need_open_cl_1, valve := "DB_TST".Valve_1, TIME_Opening := "Time_Opening_cl_1", TIME_Closing := "Time_Closing_cl_1", CMD_Open_Out => "PLC_Signals_DB".DO_1_3.Input, Alarm_Out => "DB_TST".Valve_alarm_1)
   END_RUNG
   // the same network as SCL:
   "Valve"(Valve_opening := "PLC_Signals_DB".DI_1_2.Output,
           Need_open := "DB_TST".Need_open_cl_1,
           valve := "DB_TST".Valve_1,
           TIME_Opening := "Time_Opening_cl_1",
           TIME_Closing := "Time_Closing_cl_1",
           CMD_Open_Out => "PLC_Signals_DB".DO_1_3.Input,
           Alarm_Out => "DB_TST".Valve_alarm_1);
END_REGION

REGION Network 4: Клапан контроля подачи газа на основную горелку
   RUNG wire#powerrail
      "Valve"(Valve_opening := "PLC_Signals_DB".DI_1_3.Output, Need_open := "DB_TST".Need_open_cl_2, valve := "DB_TST".Valve_2, TIME_Opening := "Time_Opening_cl_2", TIME_Closing := "Time_Closing_cl_2", CMD_Open_Out => "PLC_Signals_DB".DO_1_4.Input, Alarm_Out => "DB_TST".Valve_alarm_2)
   END_RUNG
   // the same network as SCL:
   "Valve"(Valve_opening := "PLC_Signals_DB".DI_1_3.Output,
           Need_open := "DB_TST".Need_open_cl_2,
           valve := "DB_TST".Valve_2,
           TIME_Opening := "Time_Opening_cl_2",
           TIME_Closing := "Time_Closing_cl_2",
           CMD_Open_Out => "PLC_Signals_DB".DO_1_4.Input,
           Alarm_Out => "DB_TST".Valve_alarm_2);
END_REGION

REGION Network 5: MB_Comm_Load_DB
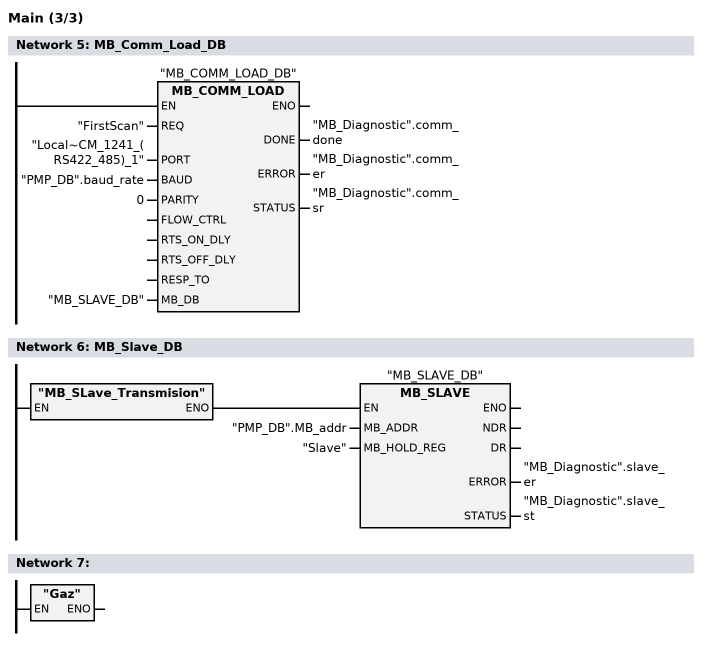
   "MB_COMM_LOAD_DB"(REQ := "FirstScan",   // MB_COMM_LOAD
                     PORT := "Local~CM_1241_(RS422_485)_1",
                     BAUD := "PMP_DB".baud_rate,
                     PARITY := 0,
                     MB_DB := "MB_SLAVE_DB",
                     DONE => "MB_Diagnostic".comm_done,
                     ERROR => "MB_Diagnostic".comm_er,
                     STATUS => "MB_Diagnostic".comm_sr);
END_REGION

REGION Network 6: MB_Slave_DB
   "MB_SLave_Transmision"(ENO => #_w1);
   IF #_w1 THEN
       "MB_SLAVE_DB"(MB_ADDR := "PMP_DB".MB_addr,   // MB_SLAVE
                     MB_HOLD_REG := "Slave",
                     ERROR => "MB_Diagnostic".slave_er,
                     STATUS => "MB_Diagnostic".slave_st);
   END_IF;
END_REGION

REGION Network 7
   RUNG wire#powerrail
      "Gaz"()
   END_RUNG
   // the same network as SCL:
   "Gaz"();
END_REGION
END_ORGANIZATION_BLOCK